// Mitsubishi GX Works2 project: 18-06-2020 Ex10 Car park   PLC: FX3G

PROGRAM MAIN
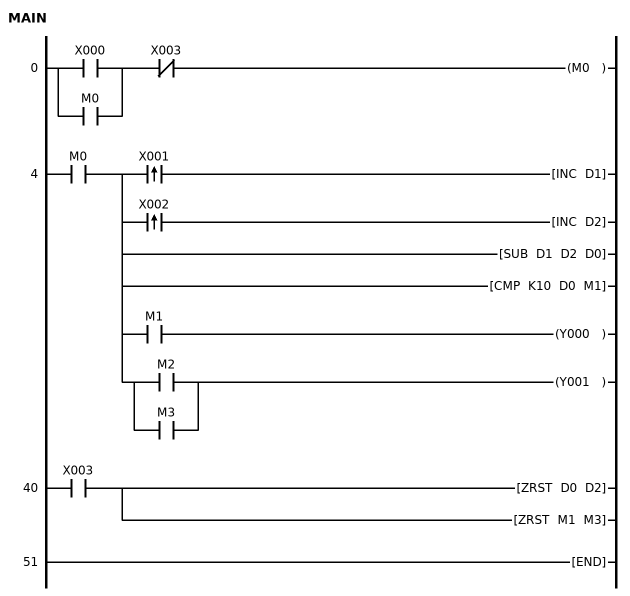
0     LD      X000
      OR      M0
      ANI     X003
      OUT     M0
4     LD      M0
      MPS
      ANDP    X001
      INC     D1
      MRD
      ANDP    X002
      INC     D2
      MPP
      SUB     D1 D2 D0
      CMP     K10 D0 M1
      MPS
      AND     M1
      OUT     Y000
      MPP
      LD      M2
      OR      M3
      ANB
      OUT     Y001
40    LD      X003
      ZRST    D0 D2
      ZRST    M1 M3
51    END
END_PROGRAM
